Fanuc KAREL source: ko00084.KL

-- PROVISIONAL review KL for V1013-1; original PC SHA256 64eefc54aa234fb1cf723a990372ee7ae6247be7d11f12f629cbb6d47c698388
-- Incomplete behavior may be omitted. Consult companion uncertainty JSON. Do not deploy.
PROGRAM KO00084
%NOLOCKGROUP
BEGIN
  -- UNRESOLVED_PC offsets 5-12; opcodes 9D,23
  -- UNRESOLVED_PC offsets 17-66; opcodes 27,27,49,7E,AD,22,1C,22,31,7E,4A
  -- UNRESOLVED_PC offsets 71-75; opcodes 7F
END KO00084
